PROGRAM p06_frontDetection
VAR
	S0: BOOL;
	S1: BOOL;
	L0: BOOL;
	L1: BOOL;
	L2: BOOL;
	PositiveEdge: R_TRIG;
	NegativeEdge: F_TRIG;		
	PositiveFrontExpr: R_TRIG;
END_VAR

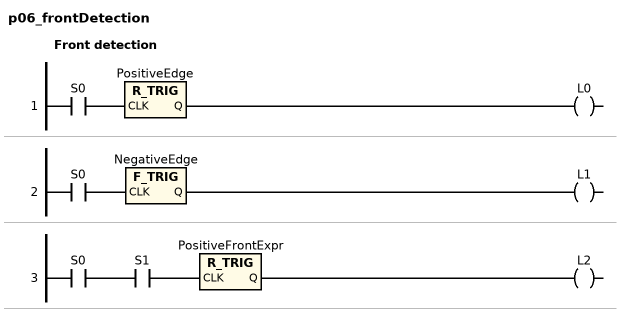
// NETWORK 1: Front detection
PositiveEdge(CLK := S0); // R_TRIG
L0 := PositiveEdge.Q;

// NETWORK 2
NegativeEdge(CLK := S0); // F_TRIG
L1 := NegativeEdge.Q;

// NETWORK 3
PositiveFrontExpr(CLK := S0 AND S1); // R_TRIG
L2 := PositiveFrontExpr.Q;

END_PROGRAM

(* stored: Version 1.1.0.1, ProductVersion 3.1.4024.13
   POU p06_frontDetection: Id {3903a342-f770-418a-9e84-020d824c4672}, SpecialFunc None *)
